FUNCTION F_LogError  
VAR_INPUT
    Message : T_MaxString;
END_VAR

ADSLOGSTR(
    msgCtrlMask := ADSLOG_MSGTYPE_STRING OR ADSLOG_MSGTYPE_ERROR OR ADSLOG_MSGTYPE_LOG,
    msgFmtStr := Message,
    strArg := '');

END_FUNCTION

(* stored: Version 1.1.0.1, ProductVersion 3.1.4024.3
   POU F_LogError: Id {a0934867-1093-02ce-1949-2db735b0211f}, SpecialFunc None *)
